// Mitsubishi GX Works2 project: tanque2   PLC: FX3U/FX3UC
// Configuração Modbus RTU

PROGRAM MAIN
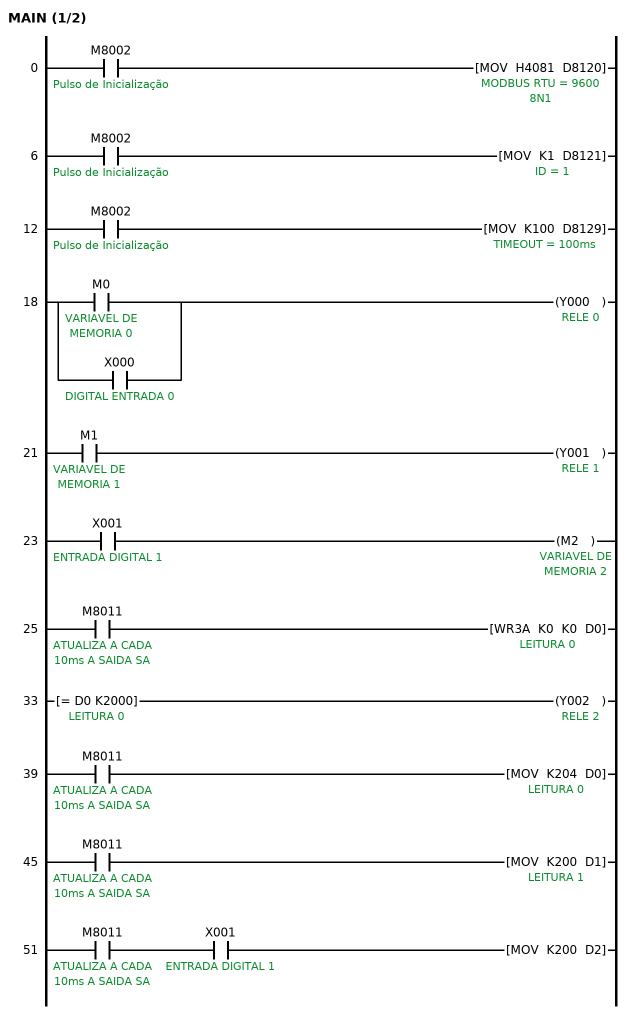
0     LD      M8002  ; Pulso de Inicialização
      MOV     H4081 D8120  ; MODBUS RTU = 9600 8N1
6     LD      M8002  ; Pulso de Inicialização
      MOV     K1 D8121  ; ID = 1
12    LD      M8002  ; Pulso de Inicialização
      MOV     K100 D8129  ; TIMEOUT = 100ms
18    LD      M0  ; VARIAVEL DE MEMORIA 0
      OR      X000  ; DIGITAL ENTRADA 0
      OUT     Y000  ; RELE 0
21    LD      M1  ; VARIAVEL DE MEMORIA 1
      OUT     Y001  ; RELE 1
23    LD      X001  ; ENTRADA DIGITAL 1
      OUT     M2  ; VARIAVEL DE MEMORIA 2
25    LD      M8011  ; ATUALIZA A CADA 10ms A SAIDA SA
      WR3A    K0 K0 D0  ; LEITURA 0
33    LD=     D0 K2000  ; LEITURA 0
      OUT     Y002  ; RELE 2
39    LD      M8011  ; ATUALIZA A CADA 10ms A SAIDA SA
      MOV     K204 D0
45    LD      M8011  ; ATUALIZA A CADA 10ms A SAIDA SA
      MOV     K200 D1  ; LEITURA 1
51    LD      M8011  ; ATUALIZA A CADA 10ms A SAIDA SA
      AND     X001  ; ENTRADA DIGITAL 1
      MOV     K200 D2
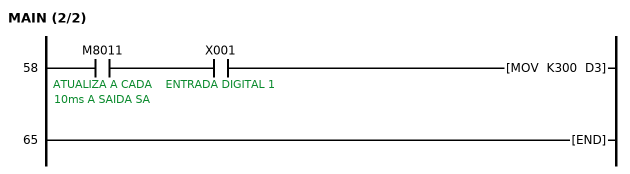
58    LD      M8011  ; ATUALIZA A CADA 10ms A SAIDA SA
      AND     X001  ; ENTRADA DIGITAL 1
      MOV     K300 D3
65    END
END_PROGRAM
